Staubli VAL3: unSelectItem.pgx

program unSelectItem()
  local string l_sEvent
  local num i
  local num l_nSize
begin
//  // remove all the comments
//  call trajType:getSizeItem(false,l_nSize)
//  for i=0 to (l_nSize-1)
//    // get all the items
//    call trajType:getTrajItem(l_tTraj,i)
//    if find(l_tTraj.comment,"#")!=-1
//      // look for the select item
//      l_tTraj.comment=right(l_tTraj.comment,len(l_tTraj.comment)-1)
//      call trajType:setTrajItem(l_tTraj,i)
//    endIf
//  endFor
end
